TYPE HMIMovementInterface :
STRUCT
	MovementSettingLines	:	ARRAY [1..3] of HMISettingLineInterface;
END_STRUCT
END_TYPE

(* stored: Version 1.1.0.1
   DUT HMIMovementInterface: Id {c32c9642-4143-4c0e-a0a1-1f71cee961ae} *)
